// TIA Portal V19 export
DATA_BLOCK "PRINTING DATA"   // DB133
{ S7_Optimized_Access := 'FALSE' }
   VAR
      "LINE 1" : String[80] := '                          M/S PHARMAFORCE LAB UNIT-II                       ';
      "LINE 2" : String[80] := '                 MFG BY : KOTHARI PHARMA TECHNOLOGIES  PVT LTD              ';
      "LINE 3" : String[80] := ' -------------------------------------------------------------------------------';
      "LINE 4" : String[80] := '                                     CIP SKID                                 ';
      "LINE 5" : String[80] := ' -------------------------------------------------------------------------------';
      "LINE 6" : String[80] := '    /  /              RINSE-1,RINSE-2, FINAL RINSE-1 PARAMETER    ';
      "LINE 7" : String[80] := ' -------------------------------------------------------------------------------';
      "LINE 8" : String[80] := '  PARAMETER                        SET VALUE';
      "LINE 9" : String[80] := '                                   RINSE-1          RINSE-2          F_RINSE-1';
      "LINE 10" : String[80] := '  HEATING TEMPERATURE  ';
      "LINE 11" : String[80] := '  CLEANING TIME ';
      "LINE 12" : String[80] := '  RECIRCULATION TIME ';
      "LINE 13" : String[80] := '  DRAIN TIME';
      "LINE 14" : String[80] := '  PUMP CASING DRAIN TIME ';
      "LINE 15" : String[80] := '  FWD PUMP HEATING RPM ';
      "LINE 16" : String[80] := '  FWD PUMP CLEANING RPM ';
      "LINE 17" : String[80];
      "LINE 18" : String[80] := ' -------------------------------------------------------------------------------';
      "LINE 19" : String[80] := '    /  /              ALKALI / ACID PARAMETER ';
      "LINE 20" : String[80] := ' -------------------------------------------------------------------------------';
      "LINE 21" : String[80] := '  PARAMETER                             SET VALUE                 ';
      "LINE 22" : String[80] := '  HEATING TEMPERATURE  ';
      "LINE 23" : String[80] := '  CLEANING TIME ';
      "LINE 24" : String[80] := '  RECIRCULATION TIME ';
      "LINE 25" : String[80] := '  DRAIN TIME';
      "LINE 26" : String[80] := '  PUMP CASING DRAIN TIME ';
      "LINE 27" : String[80] := '  FWD PUMP HEATING RPM ';
      "LINE 28" : String[80] := '  FWD PUMP CLEANING RPM ';
      "LINE 29" : String[80] := '  BEFORE CLEANING PH LOW ';
      "LINE 30" : String[80] := '  BEFORE CLEANING PH HIGH ';
      "LINE 31" : String[80] := '  AFTER CLEANING PH LOW ';
      "LINE 32" : String[80] := '  AFTER CLEANING PH HIGH ';
      "LINE 33" : String[80];
      "LINE 34" : String[80] := ' -------------------------------------------------------------------------------';
      "LINE 35" : String[80] := '    /  /              FINAL RINSE-2 PARAMETER    ';
      "LINE 36" : String[80] := ' -------------------------------------------------------------------------------';
      "LINE 37" : String[80] := '  PARAMETER                            SET VALUE                   ';
      "LINE 38" : String[80] := '  HEATING TEMPERATURE  ';
      "LINE 39" : String[80] := '  CLEANING TIME ';
      "LINE 40" : String[80] := '  RECIRCULATION TIME ';
      "LINE 41" : String[80] := '  DRAIN TIME';
      "LINE 42" : String[80] := '  PUMP CASING DRAIN TIME ';
      "LINE 43" : String[80] := '  FWD PUMP HEATING RPM ';
      "LINE 44" : String[80] := '  FWD PUMP CLEANING RPM ';
      "LINE 45" : String[80] := '  CONDUCTIVITY ';
      "LINE 46" : String[80];
      "LINE 47" : String[80];
      AL1 : String[80] := '      :  :        EMERGENCY PRESSED ';
      AL2 : String[80] := '      :  :        POWER FAIL ';
      AL3 : String[80] := '      :  :        FORWARD PUMP TRIP';
      AL4 : String[80] := '      :  :        RETURN PUMP TRIP';
      AL5 : String[80] := '      :  :        ALKALI LEVEL IS LOW';
      AL6 : String[80] := '      :  :        ACID LEVEL IS LOW';
      AL7 : String[80] := '      :  :        PURE WATER LEVLE IS LOW ';
      AL8 : String[80] := '      :  :        SOFTWATER LEVLE IS LOW ';
      AL9 : String[80] := '      :  :        AIR FAIL';
      AL10 : String[80] := '      :  :        FORWARD LIMIT SWITCH IS UNHEALTHY';
      AL11 : String[80] := '      :  :        RETURN LIMIT SWITCH IS UNHEALTHY';
      AL12 : String[80];
      PV1 : String[80] := ' -------------------------------------------------------------------------------';
      PV2 : String[80] := '    /  /              PRESENT VALUES    ';
      PV3 : String[80] := ' -------------------------------------------------------------------------------';
      PV4 : String[80] := '                     TEMP           PUMP-1_RPM           PH          CON ';
      PV5 : String[80] := '      :  :        ';
      BLANK : String[80] := '.                                                            ';
      FOOTER1 : String[80] := '  DONE BY :                                  CHECKED BY :                  ';
   END_VAR
BEGIN
END_DATA_BLOCK
